TYPE ST_Wago750495_Write_1 :
STRUCT
	b_EnableRegisterComm		: BOOL;
	e_statusQuery				: eWago750495_StatDataID; //0: status L1, 1: status L2, 2: Status L3, 3: Status IO Module			
END_STRUCT
END_TYPE

(* stored: Version 1.1.0.1, ProductVersion 3.1.4024.12
   DUT ST_Wago750495_Write_1: Id {2fcf416f-6a28-4340-b0e7-3c8df120881f} *)
